(* CODESYS project tcprocess.library
   Company: TcNexa
   DefaultNamespace: TcNexa_Components_TcProcess
   Version: 2.0.0
   Placeholder: TcProcess
   Author: ATI Software Engineering
   Description: This library serves as a valuable resource for managing reusable components within your automation projects
   Title: TcProcess

Project tree, tasks and I/O mapping:
  libraries: Tc2_Standard, * (Beckhoff Automation GmbH); Tc2_System, * (Beckhoff Automation GmbH); Tc3_Module, * (Beckhoff Automation GmbH)
  Method Reponse/
    function block FB_MethodResponse [ST]: _clear, busy, error, errorDescription, message, copyFrom, setBusy, setFail, setPass
  Step/
    function block FB_Step [ST]: actual, inc, init, set
  Tests/
    program PRG_TEST [ST]
  Version/
    global variables Global_Version
*)

// Version/Global_Version
{attribute 'TcGenerated'}
{attribute 'no-analysis'}
{attribute 'linkalways'}
// This function has been automatically generated from the project information.
VAR_GLOBAL CONSTANT
	{attribute 'const_non_replaced'}
	stLibVersion_TcProcess : ST_LibVersion := (iMajor := 2, iMinor := 0, iBuild := 0, iRevision := 0, nFlags := 0, sVersion := '2.0.0');
END_VAR

// Method Reponse/FB_MethodResponse
FUNCTION_BLOCK FB_MethodResponse
VAR
	_busy				: BOOL;				// Indicates if the method call is in progress
	_error				: BOOL;				// Indicates if the method call failed
	_message			: STRING(255);
	_errorDescription	: STRING(255);		// Information to show to the user
END_VAR

METHOD PROTECTED _clear
VAR_INPUT
END_VAR
_busy:= FALSE;
_error:= FALSE;
_message:= '';
_errorDescription:= '';
END_METHOD

PROPERTY PUBLIC busy : BOOL
GET
busy:= _busy;
END_GET
END_PROPERTY

PROPERTY PUBLIC error : BOOL
GET
error:= _error;
END_GET
END_PROPERTY

PROPERTY PUBLIC errorDescription : STRING(255)
GET
errorDescription:= _errorDescription;
END_GET
END_PROPERTY

PROPERTY PUBLIC message : STRING(255)
GET
message:= _message;
END_GET
END_PROPERTY

METHOD PUBLIC copyFrom
VAR_INPUT
	Response		: FB_MethodResponse;
END_VAR
_busy:= Response.busy;
_error:= Response.error;
_message:= Response.message;
_errorDescription:= Response.errorDescription;
END_METHOD

METHOD PUBLIC setBusy
VAR_INPUT
	message	 	: STRING(255);
END_VAR
_clear();

_busy:= TRUE;
_message:= message;
END_METHOD

METHOD PUBLIC setFail
VAR_INPUT
	message				: STRING(255);
	description			: STRING(255);
END_VAR
_clear();

_error:= TRUE;
_message:= message;
_errorDescription:= description;
END_METHOD

METHOD PUBLIC setPass
VAR_INPUT
END_VAR
_clear();
END_METHOD

END_FUNCTION_BLOCK

// Step/FB_Step
FUNCTION_BLOCK FB_Step
VAR
	_actual						: INT:= -1;
END_VAR

PROPERTY PUBLIC actual : INT
GET
PUBLIC 
VAR
END_VAR
actual:= _actual;
END_GET
END_PROPERTY

METHOD PUBLIC inc
VAR
END_VAR
_actual:= _actual + 1;
END_METHOD

METHOD PUBLIC init
VAR_INPUT
END_VAR
_actual:= 0;
END_METHOD

METHOD PUBLIC set
VAR_INPUT
	target	: INT;
END_VAR
_actual:= target;
END_METHOD

END_FUNCTION_BLOCK

// Tests/PRG_TEST
PROGRAM PRG_TEST
VAR
END_VAR

END_PROGRAM
